FUNCTION_BLOCK FB_Object_Template_ST
VAR_INPUT
	// Control variables
	Execute: BOOL;
	Ack: BOOL;
	Reset: BOOL; 
	Pause: BOOL;
	// Physical variables
	
END_VAR
VAR_OUTPUT
	//Control variables
	Ready: BOOL;
	Done: BOOL;
	//Physical Variables
	
END_VAR
VAR
	// Initial conditions
	IC: BOOL := TRUE;
END_VAR

END_FUNCTION_BLOCK

(* stored: Version 1.1.0.1, ProductVersion 3.1.4024.6
   POU FB_Object_Template_ST: Id {bebdeb7d-5ec3-4d18-ae03-9d3a3c412779}, SpecialFunc None *)
